// Mitsubishi GX Works2 project: may_son_new   PLC: FX3U/FX3UC

PROGRAM MAIN
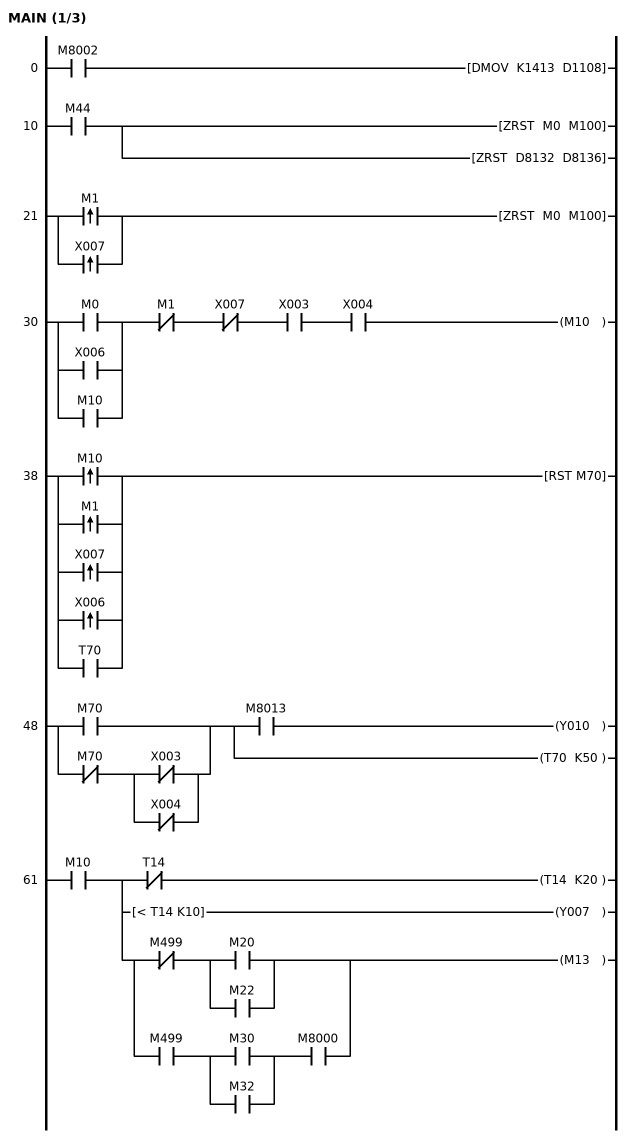
0     LD      M8002
      DMOV    K1413 D1108
10    LD      M44
      ZRST    M0 M100
      ZRST    D8132 D8136
21    LDP     M1
      ORP     X007
      ZRST    M0 M100
30    LD      M0
      OR      X006
      OR      M10
      ANI     M1
      ANI     X007
      AND     X003
      AND     X004
      OUT     M10
38    LDP     M10
      ORP     M1
      ORP     X007
      ORP     X006
      OR      T70
      RST     M70
48    LD      M70
      LDI     M70
      LDI     X003
      ORI     X004
      ANB
      ORB
      MPS
      AND     M8013
      OUT     Y010
      MPP
      OUT     T70 K50
61    LD      M10
      MPS
      ANI     T14
      OUT     T14 K20
      MRD
      AND<    T14 K10
      OUT     Y007
      MPP
      LDI     M499
      LD      M20
      OR      M22
      ANB
      LD      M499
      LD      M30
      OR      M32
      ANB
      AND     M8000
      ORB
      ANB
      OUT     M13
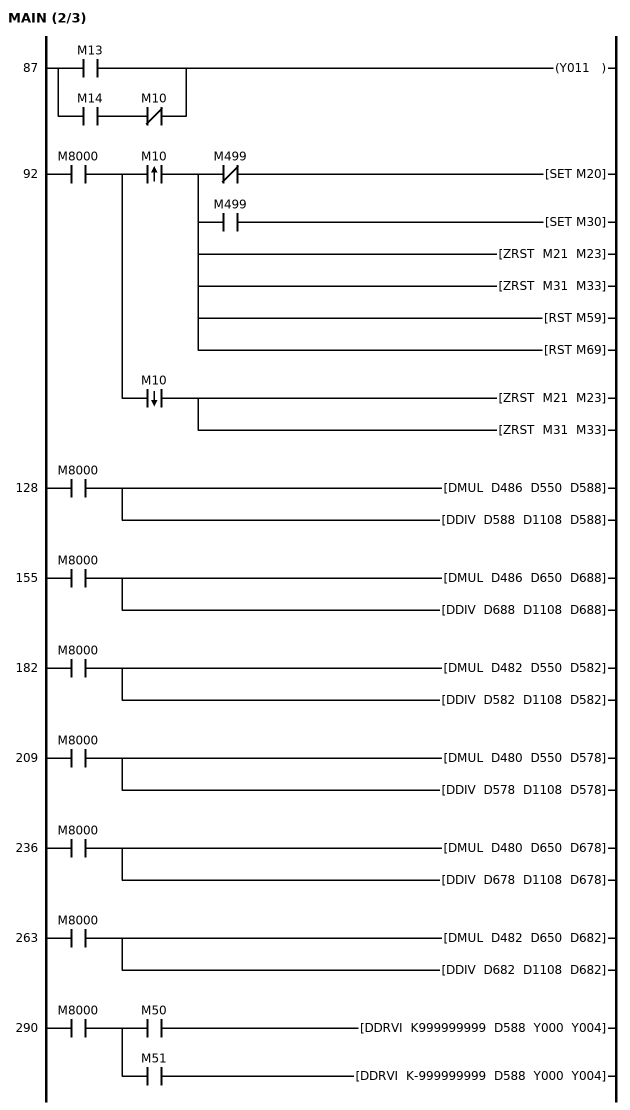
87    LD      M13
      LD      M14
      ANI     M10
      ORB
      OUT     Y011
92    LD      M8000
      MPS
      ANDP    M10
      MPS
      ANI     M499
      SET     M20
      MRD
      AND     M499
      SET     M30
      MPP
      ZRST    M21 M23
      ZRST    M31 M33
      RST     M59
      RST     M69
      MPP
      ANDF    M10
      ZRST    M21 M23
      ZRST    M31 M33
128   LD      M8000
      DMUL    D486 D550 D588
      DDIV    D588 D1108 D588
155   LD      M8000
      DMUL    D486 D650 D688
      DDIV    D688 D1108 D688
182   LD      M8000
      DMUL    D482 D550 D582
      DDIV    D582 D1108 D582
209   LD      M8000
      DMUL    D480 D550 D578
      DDIV    D578 D1108 D578
236   LD      M8000
      DMUL    D480 D650 D678
      DDIV    D678 D1108 D678
263   LD      M8000
      DMUL    D482 D650 D682
      DDIV    D682 D1108 D682
290   LD      M8000
      MPS
      AND     M50
      DDRVI   K999999999 D588 Y000 Y004
      MPP
      AND     M51
      DDRVI   K-999999999 D588 Y000 Y004
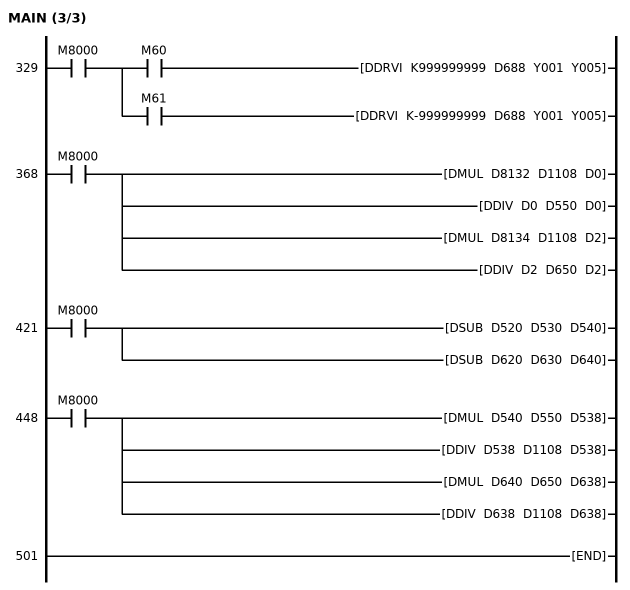
329   LD      M8000
      MPS
      AND     M60
      DDRVI   K999999999 D688 Y001 Y005
      MPP
      AND     M61
      DDRVI   K-999999999 D688 Y001 Y005
368   LD      M8000
      DMUL    D8132 D1108 D0
      DDIV    D0 D550 D0
      DMUL    D8134 D1108 D2
      DDIV    D2 D650 D2
421   LD      M8000
      DSUB    D520 D530 D540
      DSUB    D620 D630 D640
448   LD      M8000
      DMUL    D540 D550 D538
      DDIV    D538 D1108 D538
      DMUL    D640 D650 D638
      DDIV    D638 D1108 D638
501   END
END_PROGRAM
